TYPE ST_ProductPar :
STRUCT
	PlaceHolder			: BOOL;
END_STRUCT
END_TYPE

(* stored: Version 1.1.0.1, ProductVersion 3.1.4020.12
   DUT ST_ProductPar: Id {bc862ad1-6b85-4b6f-ae3b-b23b7db05634} *)
